PROGRAM MAIN
VAR CONSTANT
	//hlavni stavovy automat
	WAITING_FOR_START : USINT := 0;
	INIT_ROBOTS : USINT := 1; //inicializace handleru plechovek i velkeho robota
	INIT_ROBOTS_WAIT : USINT := 2; //cekaci stav, protoze pouzivam casovac
	GRAB_BOX : USINT := 3;
	GRAB_BOX_WAIT : USINT := 4;
	PUT_BOX : USINT := 5;
	PUT_BOX_WAIT : USINT := 6;
	DRIVE_BOX_TO_HANDLER : USINT := 7;
	HANDLE_CAN1 : USINT := 8;
	HANDLE_CAN1_WAIT : USINT := 9;
	HANDLE_CAN2 : USINT := 10;
	HANDLE_CAN2_WAIT : USINT := 11;
	HANDLE_CAN3 : USINT := 12;
	HANDLE_CAN3_WAIT : USINT := 13;
	CANS_HANDLED : USINT := 14;
	STORAGE_INIT : USINT := 15;
	STORAGE_INIT_WAIT : USINT := 16;
	GET_BOX_STORE : USINT := 17;
	GET_BOX_STORE_WAIT : USINT := 18;
	STORAGE_HANDLER_TO_BOX : USINT := 19;
	STORAGE_HANDLER_TO_BOX_WAIT: USINT := 20;
	LOAD_BOX : USINT := 21;
	LOAD_BOX_WAIT : USINT := 22;
	DRIVE_BOX_TO_STORE : USINT := 23;
	DRIVE_BOX_TO_STORE_WAIT : USINT := 24;
	BOX_UNLOAD : USINT := 25;
	BOX_UNLOAD_WAIT : USINT := 26;
	LAY_BOX : USINT := 27;
	STORING_DONE : USINT := 28;
END_VAR

VAR
	MainState : USINT := WAITING_FOR_START;
	StartProcess : BOOL := FALSE;
	CanSpeed : WORD := 1900;
	ConvSpeed : WORD := 2800;
	BoxAtTheEnd : BOOL := FALSE;
	TON_DelayCycle : TON;
	x : ARRAY [0..10] OF WORD := [25580, 23000, 20420, 17845, 15260, 12700, 10120, 7520, 4940, 2380, 750];
	y : ARRAY [0..5] OF WORD := [23750, 19142, 14535, 9927, 5318, 710];
	//FirstBoxDriven : BOOL := FALSE;
	BoxesStored : USINT := 0;
	ID : ARRAY [0..5] OF USINT := [2,5,6,3,9,4];
	P_RegulatorX : P_regulator;
	P_RegulatorY : P_regulator;
	yPosition : WORD := 0;
	xPosition : WORD := 0;
	RoboticArmStart : BOOL := FALSE;
	CentralStop : BOOL := FALSE;
END_VAR


IOmap(); //namapuj vstupy a vystupy
IF CentralStop THEN
	IO.ConvBoxEnable := 0;
	IO.ConvCanEnable := 0;
	IO.StorageSupportEnable := 0;
	IO.StorageCarriageEnable := 0;
	IO.StorageSupportEnable := 0;
END_IF

CASE MainState OF
	WAITING_FOR_START:
		IF StartProcess THEN
			MainState := INIT_ROBOTS;
		END_IF
		
	INIT_ROBOTS:
		IO.HandlingProgram := IO.RoboticArmProgram := 0;
		IO.HandlingStartCycle := IO.RoboticArmStartCycle := 1;
		TON_DelayCycle(IN := TRUE, PT := T#1S);
		IF TON_DelayCycle.Q THEN
			TON_DelayCycle(IN := 0);
			IF NOT IO.RoboticArmMoving AND NOT IO.HandlingMoving THEN
				IO.HandlingStartCycle := IO.RoboticArmStartCycle := 0;
				MainState := INIT_ROBOTS_WAIT;
			END_IF
		END_IF
		
	INIT_ROBOTS_WAIT:
		TON_DelayCycle(IN := TRUE, PT := T#1S);
		IF TON_DelayCycle.Q THEN
			TON_DelayCycle(IN := 0); 
			MainState := GRAB_BOX;
		END_IF
		
	GRAB_BOX:
		IO.RoboticArmProgram := 1;
		IO.RoboticArmStartCycle := 1;
		TON_DelayCycle(IN := TRUE, PT := T#1S);
		IF TON_DelayCycle.Q THEN
			TON_DelayCycle(IN := 0);
			IF NOT IO.RoboticArmMoving THEN
				IO.RoboticArmStartCycle := 0;
				MainState := GRAB_BOX_WAIT;
			END_IF
		END_IF
		
	GRAB_BOX_WAIT:
		TON_DelayCycle(IN := TRUE, PT := T#1S);
		IF TON_DelayCycle.Q THEN
			TON_DelayCycle(IN := 0);
			MainState := PUT_BOX;
		END_IF
	
	PUT_BOX:
		IO.RoboticArmProgram := 2;
		IO.RoboticArmStartCycle := 1;
		TON_DelayCycle(IN := TRUE, PT := T#1S);
		IF TON_DelayCycle.Q THEN 
			TON_DelayCycle(IN := 0);
			IF NOT IO.RoboticArmMoving THEN
				IO.RoboticArmStartCycle := 0;
				MainState := PUT_BOX_WAIT;
			END_IF
			
		END_IF
		
	PUT_BOX_WAIT:
		TON_DelayCycle(IN := TRUE, PT := T#1S);
		IF TON_DelayCycle.Q THEN
			TON_DelayCycle(IN := 0);
			MainState := DRIVE_BOX_TO_HANDLER;
		END_IF
		
	DRIVE_BOX_TO_HANDLER:
		
		IF IO.SensorBoxHandling THEN
			IO.ConvBoxEnable := 0;
			MainState := HANDLE_CAN1;
		ELSE
			IO.ConvBoxEnable := 1;
		END_IF
		
		
	HANDLE_CAN1:
		IO.HandlingProgram := 1;
		IO.HandlingStartCycle := 1;
		TON_DelayCycle(IN := TRUE, PT := T#1S);
		IF TON_DelayCycle.Q THEN
			TON_DelayCycle(IN := 0);
			IF NOT IO.HandlingMoving THEN
				IO.HandlingStartCycle := 0; 
				MainState := HANDLE_CAN1_WAIT;
			END_IF
		END_IF
		
	HANDLE_CAN1_WAIT:
		TON_DelayCycle(IN := TRUE, PT := T#1S);
		IF TON_DelayCycle.Q THEN
			TON_DelayCycle(IN := 0); 
			MainState := HANDLE_CAN2;
		END_IF
		
	HANDLE_CAN2:
		TON_DelayCycle(IN := TRUE, PT := T#1S);
		IO.HandlingProgram := 2;
		IO.HandlingStartCycle := 1;
		IF TON_DelayCycle.Q THEN
			TON_DelayCycle(IN := 0);
			IF NOT IO.HandlingMoving THEN
				IO.HandlingStartCycle := 0;
				MainState := HANDLE_CAN2_WAIT;
			END_IF
		END_IF
		
	HANDLE_CAN2_WAIT:
		TON_DelayCycle(IN := TRUE, PT := T#1S);
		IF TON_DelayCycle.Q THEN
			TON_DelayCycle(IN := 0); 
			MainState := HANDLE_CAN3;
		END_IF
		
	HANDLE_CAN3:
		TON_DelayCycle(IN := TRUE, PT := T#1S);
		IO.HandlingProgram := 3;
		IO.HandlingStartCycle := 1;
		IF TON_DelayCycle.Q THEN
			TON_DelayCycle(IN := 0);
			IF NOT IO.HandlingMoving THEN
				IO.HandlingStartCycle := 0; 
				MainState := HANDLE_CAN3_WAIT;
			END_IF
		END_IF
		
	HANDLE_CAN3_WAIT:
		TON_DelayCycle(IN := TRUE, PT := T#1S);
		IF TON_DelayCycle.Q THEN
			TON_DelayCycle(IN := 0);
			MainState := CANS_HANDLED;
		END_IF	
	
	CANS_HANDLED:
		MainState := GET_BOX_STORE;
		IO.ConvBoxEnable := 1;
	
	STORAGE_INIT:
		TON_DelayCycle(IN := TRUE, PT := T#1S);
		
		P_RegulatorX.SetpointPos := 750;
		P_RegulatorY.SetpointPos := 1100;
		
		IF TON_DelayCycle.Q THEN
			TON_DelayCycle(IN := 0);
			IF NOT IO.StorageCarriageMoving AND NOT IO.StorageSupportMoving THEN
				
				MainState := STORAGE_INIT_WAIT;
			END_IF
		
		END_IF
		
	STORAGE_INIT_WAIT:
		TON_DelayCycle(IN := TRUE, PT := T#1S);
		IF TON_DelayCycle.Q THEN
			TON_DelayCycle(IN := 0); 
			MainState := GET_BOX_STORE;
		END_IF
		
	GET_BOX_STORE:
		IO.StorageCarriageEnable := IO.StorageSupportEnable := 1;
		IF IO.SensorBoxStoring THEN
			TON_DelayCycle(IN := TRUE, PT := T#1S);
			P_RegulatorX.SetpointPos := 750;
			P_RegulatorY.SetpointPos := 1100;	
			IF TON_DelayCycle.Q THEN
					IF NOT IO.StorageSupportMoving AND NOT IO.StorageCarriageMoving THEN
						
						MainState := GET_BOX_STORE_WAIT;
					END_IF
			END_IF
		END_IF
		
	GET_BOX_STORE_WAIT:
		TON_DelayCycle(IN := TRUE, PT := T#1S);
		IF TON_DelayCycle.Q THEN
			TON_DelayCycle(IN := 0); 
			
			MainState := STORAGE_HANDLER_TO_BOX;
		END_IF
		
	STORAGE_HANDLER_TO_BOX:
		TON_DelayCycle(IN := TRUE, PT := T#2S);
		IF TON_DelayCycle.Q THEN
			P_RegulatorY.SetpointPos := 2100;
			IO.StorageLoad := 1;
			MainState := STORAGE_HANDLER_TO_BOX_WAIT;
		END_IF
	
	STORAGE_HANDLER_TO_BOX_WAIT:
		TON_DelayCycle(IN := TRUE, PT := T#2S);
		IF TON_DelayCycle.Q THEN
			
			TON_DelayCycle(IN := FALSE);
			MainState := LOAD_BOX;
		END_IF
		
	LOAD_BOX:
		TON_DelayCycle(IN := TRUE, PT := T#2S);
		IF TON_DelayCycle.Q THEN
			TON_DelayCycle(IN := FALSE);
			IO.StorageLoad := 0;
			MainState := LOAD_BOX_WAIT;
		END_IF
		
	LOAD_BOX_WAIT:
		TON_DelayCycle(IN := TRUE, PT := T#2S);
		IF TON_DelayCycle.Q THEN
			TON_DelayCycle(IN := FALSE);
			MainState := DRIVE_BOX_TO_STORE;
		END_IF
	
		
	DRIVE_BOX_TO_STORE: 
		TON_DelayCycle(IN := TRUE, PT := T#1S);
		IF TON_DelayCycle.Q THEN
			TON_DelayCycle(IN := FALSE);
				P_RegulatorX.SetpointPos := x[ID[BoxesStored]];
				P_RegulatorY.SetpointPos := y[BoxesStored] + 400;
			MainState := DRIVE_BOX_TO_STORE_WAIT; 
		END_IF
		
	DRIVE_BOX_TO_STORE_WAIT:
		TON_DelayCycle(IN := TRUE, PT := T#1S);
		IF TON_DelayCycle.Q THEN
			TON_DelayCycle(IN := FALSE);
			MainState := BOX_UNLOAD;
		END_IF
		
	BOX_UNLOAD: 
		TON_DelayCycle(IN := TRUE, PT := T#1S);
		IF TON_DelayCycle.Q THEN
			IF NOT IO.StorageCarriageMoving AND NOT IO.StorageSupportMoving THEN
				TON_DelayCycle(IN := FALSE);
				IO.StorageUnload := 1;
				MainState := BOX_UNLOAD_WAIT;
			END_IF
		END_IF
	BOX_UNLOAD_WAIT:
		TON_DelayCycle(IN := TRUE, PT := T#1S);
		IF TON_DelayCycle.Q THEN
				TON_DelayCycle(IN := FALSE);
				MainState := LAY_BOX;
				P_RegulatorY.SetpointPos := P_RegulatorY.SetpointPos - 400;
		END_IF
		
	LAY_BOX:
		TON_DelayCycle(IN := TRUE, PT := T#1S);
		IF TON_DelayCycle.Q THEN
			IF NOT IO.StorageCarriageMoving AND NOT IO.StorageSupportMoving THEN
				TON_DelayCycle(IN := FALSE);
				IO.StorageUnload := 0;
				IF BoxesStored < 5 THEN
					MainState := GRAB_BOX;
					BoxesStored := BoxesStored + 1;
				ELSE
					MainState := STORING_DONE;
				END_IF
			END_IF 
			
		END_IF
		
END_CASE

IF IO.SensorBoxHandled THEN
	BoxAtTheEnd := TRUE;
END_IF

//maly dopravnik
IO.ConvCanSpeed := CanSpeed;
IO.ConvCanForward := TRUE;
IO.ConvCanEnable := NOT IO.SensorCanHandling AND MainState > WAITING_FOR_START;
StartProcess := FALSE;

//velky dopravnik
IO.ConvBoxSpeed := ConvSpeed;
IO.ConvBoxForward := TRUE;

//zakladaci dopravnik
IO.ConvLoadSpeed := ConvSpeed;
IO.ConvLoadForward := TRUE;
IO.ConvLoadEnable := BoxAtTheEnd AND NOT IO.SensorBoxStoring;

P_RegulatorX(CurrentPos := IO.StorageSupportPosition, DecelerationLength := 15000);
IO.StorageSupportSpeed := REAL_TO_WORD(P_RegulatorX.Speed);
IO.StorageSupportForward := P_RegulatorX.MoveForward;
IO.StorageSupportBackward := P_RegulatorX.MoveBackward;

P_RegulatorY(CurrentPos := IO.StorageCarriagePosition, DecelerationLength := 17000);
IO.StorageCarriageSpeed := REAL_TO_WORD(P_RegulatorY.Speed);
IO.StorageCarriageForward := P_RegulatorY.MoveForward;
IO.StorageCarriageBackward := P_RegulatorY.MoveBackward;

END_PROGRAM

(* stored: Version 1.1.0.1, ProductVersion 3.1.4024.15
   POU MAIN: Id {ea4da398-e343-4c9d-b28f-f0096319345c}, SpecialFunc None *)
